PROGRAM mySAFETY
VAR
	ResetReq	: bool;
	bPlc2TsErrAck AT %Q* : BOOL;
	bPlc2TsRestart AT %Q* : BOOL;
	bPlc2TsSTO AT %Q* : BOOL;
	bInit: BOOL;
	bTsToPlcEstopState AT %I* : BOOL := TRUE;
	bPlc2TsRun AT %Q* : BOOL := TRUE;
	ranint : INT;
	ranbool : BOOL;
	ranbool2 : bool;
END_VAR


bPlc2TsErrAck := FALSE;
IF NOT bInit THEN
	bInit := TRUE;
	bPlc2TsErrAck := TRUE;
END_IF

IF NOT bTsToPlcEstopState THEN
	PLCAxisEnable := FALSE;
END_IF

IF GVL_IO.bEstopPB = FALSE THEN
	GVL_IO.bAceOn := FALSE;
 	GVL_IO.bSprayOn := FALSE;
	GVL_IO.iTrunSig := 0;
END_IF

IF GVL_HMI.ManualMode AND GVL_SAF.DeadmanEnable AND GVL_SAF.EStopOK THEN
	
	GVL_HMI.EnableAll := 1;
	PLCAxisEnable := 1;
	KM1_ContactorOn := 1;
	KM2_ContactorOn := 1;
	
ELSIF GVL_HMI.ManualMode THEN//TEMP REMOVE THIS
	
	GVL_HMI.EnableAll := 1;
	KM1_ContactorOn := 1;
	KM2_ContactorOn := 1;
	
ELSIF GVL_HMI.AutoMode AND GVL_SAF.DeadmanEnable AND GVL_SAF.EStopOK THEN //REMOVE THIS LATER
	
	GVL_HMI.EnableAll := 1;
	PLCAxisEnable := 1;
	KM1_ContactorOn := 1;
	KM2_ContactorOn := 1;
	
ELSE
	
	GVL_HMI.EnableAll := 0;
	PLCAxisEnable := 0;
	KM1_ContactorOn := 0;
	KM2_ContactorOn := 0;

END_IF

(*
IF GVL_HMI.ManualMode AND GVL_SAF.DeadmanEnable AND GVL_SAF.EStopOK THEN
	
	GVL_HMI.EnableAll := 1;
	PLCAxisEnable := 1;
	KM1_ContactorOn := 1;
	KM2_ContactorOn := 1;
	
	ELSE
	
	GVL_HMI.EnableAll := 0;
	PLCAxisEnable := 0;
	KM1_ContactorOn := 0;
	KM2_ContactorOn := 0;

END_IF*)

END_PROGRAM

(* stored: Version 1.1.0.1, ProductVersion 3.1.4024.12
   POU mySAFETY: Id {842f556e-02df-400e-9a48-c0f38860887d}, SpecialFunc None *)
